TYPE TcoTixonPickVibro_Status_v_1_x_x EXTENDS TcoTixonGenericStatus : 
STRUCT
    {attribute addProperty Name "<#Separator in work position#> - i6"}
    SeparatorWorkPos : BOOL;
    {attribute addProperty Name "<#In Pick Zone#>"}
    InPickZone : BOOL;
END_STRUCT
END_TYPE

(* stored: Version 1.1.0.1, ProductVersion 3.1.4024.12
   DUT TcoTixonPickVibro_Status_v_1_x_x: Id {64c7d329-7f1f-07d3-0c7c-204fad6f1457} *)
